// TIA Portal V19 export
TYPE "ItemCommand_UDT"
   STRUCT
      SpareBool : Bool;
      SpareBool_1 : Bool;
      SpareBool_2 : Bool;
      SpareBool_3 : Bool;
      SpareBool_4 : Bool;
      SpareBool_5 : Bool;
      SpareBool_6 : Bool;
      SpareBool_7 : Bool;
      Auto : Bool;
      Man_DeAct : Bool;
      Man_Act : Bool;
      Locate : Bool;
      SV_2SelectionBit : Bool;
      SV_3SelectionBit : Bool;
      Teach : Bool;
      SpareBool_10 : Bool;
   END_STRUCT;
END_TYPE
